// TwinCAT 3 PLC project plc
// ProgramVersion: 3.1.4024.0
// libraries:
//   Tc2_Standard, * (Beckhoff Automation GmbH)
//   Tc2_System, * (Beckhoff Automation GmbH)
//   Tc3_Module, * (Beckhoff Automation GmbH)
// project tree:
//   GVLs/ IO.TcGVL
//   / PlcTask.TcTTO
//   POUs/ FB_Autoritenuta.TcPOU, MAIN.TcPOU
// real-time tasks:
//   TASK PlcTask: cycle T#10ms, priority 20, ADS port 350

CONFIGURATION plc
    RESOURCE PLC ON TwinCAT3
        TASK PlcTask(INTERVAL := T#10ms, PRIORITY := 20);
        PROGRAM MAIN WITH PlcTask : MAIN;
    END_RESOURCE
END_CONFIGURATION

// ---- GVLs/IO.TcGVL
{attribute 'qualified_only'}
VAR_GLOBAL
	bStart	:	BOOL;
	bStop	:	BOOL;
	bHOn	:	BOOL;
END_VAR

// ---- POUs/MAIN.TcPOU
PROGRAM MAIN
VAR
	autoritenuta1	:	FB_Autoritenuta;
END_VAR

autoritenuta1(start:= IO.bStart, stop:= IO.bStop , onoff=> IO.bHOn);

END_PROGRAM

// ---- POUs/FB_Autoritenuta.TcPOU
FUNCTION_BLOCK FB_Autoritenuta
VAR_INPUT
	start	:	BOOL;  // NA
	stop	:	BOOL;  // NC
END_VAR
VAR_OUTPUT
	onoff	:	BOOL;
END_VAR
VAR
	stato	:	BOOL := FALSE;
END_VAR

stato := (start OR stato) AND stop;

onoff := stato;

END_FUNCTION_BLOCK
